// TIA Portal V20 export
DATA_BLOCK "Instance_FB_HMI_DB"   // DB111
// stored: AutoNumber false, InstanceOfName FB_HMI, InstanceOfType FB
"FB_HMI"
   // VAR_INPUT
   //    Control_Screen_HMI : Word;
   //    Employee_Rework : String[6];
   //    Admin_1 : String[6];
   //    Admin_2 : String[6];
   //    Admin_3 : String[6];
   //    Admin_4 : String[6];
   //    Admin_5 : String[6];
   //    Alarm_0 : Word;
   //    Alarm_1 : Word;
   //    Alarm_2 : Word;
   // END_VAR
   // VAR_OUTPUT
   //    Alarm : Bool;
   //    Job_Mailbox : Array[0..3] of Word;
   // END_VAR
   // VAR
   //    Aux_Trigger_0 : Bool;
   //    Aux_Trigger_1 : Bool;
   //    Aux_Trigger_2 : Bool;
   //    Aux_Trigger_3 : Bool;
   //    Aux_Trigger_4 : Bool;
   //    Aux_Trigger_5 : Bool;
   //    Aux_Trigger_6 : Bool;
   //    Aux_Trigger_7 : Bool;
   //    Aux_Trigger_8 : Bool;
   //    Aux_Trigger_9 : Bool;
   //    Aux_Trigger_10 : Bool;
   //    Everybody_Can_Access : Bool;
   //    Only_Admin_Can_Access : Bool;
   //    Control_Screen : Word;
   //    Timer_Delay_Change_Screen { S7_SetPoint := 'True'} : TON_TIME;
   //    Timer_Delay_Change_Job_Mailbox { S7_SetPoint := 'True'} : TON_TIME;
   // END_VAR
BEGIN
END_DATA_BLOCK
